{attribute addProperty BoxType "EL5102-0000-0016"}
{attribute addProperty Id "ENC_Status_ChannelAT %I*ARRAY[0..1] OF ENC_Status_Channel_D7AAABA7256320ENC_Control_ChannelAT %Q*ARRAY[0..1] OF ENC_Control_Channel_C4E6260B96120WcStateAT %I*WcState_98A4DF7520.250InfoDataAT %I*InfoData_BC63D37F80100"}
{attribute addProperty CRC "1793915534"}
{attribute addProperty SizeInBites "434"}
{attribute addProperty SizeInBytes "54.25"}
TYPE EL5102_C51BD5F6 :
STRUCT
	{attribute addProperty Name "ENC_Status_Channel"}
	ENC_Status_Channel : ARRAY[0..1] OF ENC_Status_Channel_D7AAABA7;
	{attribute addProperty Name "ENC_Control_Channel"}
	ENC_Control_Channel : ARRAY[0..1] OF ENC_Control_Channel_C4E6260B;
	{attribute addProperty Name "WcState"}
	WcState : WcState_98A4DF75;
	{attribute addProperty Name "InfoData"}
	InfoData : InfoData_BC63D37F;
END_STRUCT
END_TYPE

(* stored: Version 1.2.0.0, ProductVersion 3.1.4024.9
   DUT EL5102_C51BD5F6: Id {0d03c5f3-9da5-4e52-90f4-4c73fea8dc2e} *)
